// TwinCAT 3 PLC project VFDLibraryPLC
// ProgramVersion: 3.1.4023.0
// libraries:
//   Tc2_EtherCAT, * (Beckhoff Automation GmbH)
//   Tc2_Standard, * (Beckhoff Automation GmbH)
//   Tc2_System, * (Beckhoff Automation GmbH)
//   Tc2_Utilities, * (Beckhoff Automation GmbH)
//   Tc3_Module, * (Beckhoff Automation GmbH)
//   VLT_ECAT_LIB_V1_12,1.12,Danfoss Drives
// project tree:
//   DUTs/ ST_VLTParameterData.TcDUT
//   GVLs/ GVL_HMI.TcGVL
//   / PlcTask.TcTTO
//   POUs/ FB_VLTDriveControl.TcPOU, MAIN.TcPOU
// real-time tasks:
//   TASK PlcTask: cycle T#10ms, priority 20, ADS port 350
// I/O:
//   DEVICE Device 4 (EtherCAT), AmsNetId 5.24.39.150.5.1
//     Box 1 (FC-302 VLT® Automation Drive) [FC-302 VLT® Automation Drive]
// variable links:
//   (this object) <-> Device 4 (EtherCAT)/Box 1 (FC-302 VLT® Automation Drive)
//     PlcTask Inputs/MAIN.fbDriveControl.fbDriveBasic.COMM_STATUS <-> InfoData/State
//     PlcTask Inputs/MAIN.fbDriveControl.fbDriveBasic.PCDREAD.MAIN_ACTUAL_VALUE <-> Transmit PDO Parameter/1605. Main Actual Value [%]
//     PlcTask Inputs/MAIN.fbDriveControl.fbDriveBasic.PCDREAD.MOTORCURRENT <-> Transmit PDO Parameter/1614. Motor current
//     PlcTask Inputs/MAIN.fbDriveControl.fbDriveBasic.PCDREAD.STATUS_WORD <-> Transmit PDO Parameter/1603. Status Word
//     PlcTask Outputs/MAIN.fbDriveControl.fbDriveBasic.PCDWRITE.CONTROL_WORD <-> Receive PDO Parameter/1680. Fieldbus CTW 1
//     PlcTask Outputs/MAIN.fbDriveControl.fbDriveBasic.PCDWRITE.REF_VALUE <-> Receive PDO Parameter/1682. Fieldbus REF 1

CONFIGURATION VFDLibraryPLC
    RESOURCE PLC ON TwinCAT3
        TASK PlcTask(INTERVAL := T#10ms, PRIORITY := 20);
        PROGRAM MAIN WITH PlcTask : MAIN;
    END_RESOURCE
END_CONFIGURATION

// ---- DUTs/ST_VLTParameterData.TcDUT
TYPE ST_VLTParameterData :
STRUCT
	//nType		: UINT; //1 for number 2 for string.
	nRdVal		: ULINT;
	strRdVal	: STRING;
	nWrVal		: UDINT;
	strWrVal	: STRING;
END_STRUCT
END_TYPE

// ---- GVLs/GVL_HMI.TcGVL
{attribute 'qualified_only'}
VAR_GLOBAL
	bReset		: BOOL;
	bWarning	: BOOL;
	bHandOn		: BOOL;
	bOkay		: BOOL;
	bOff		: BOOL;
	bAutoOn		: BOOL;
	bAlarm		: BOOL;
	arrParamData	: ARRAY[0..99] OF ST_VLTParameterData;
	arrParamNo		: ARRAY[0..99] OF UINT;
	nParamCount	:	INT;
	bRdParams	: BOOL;
	bRdDone		: BOOL;
	bWrParams	: BOOL;
	bWrDone		: BOOL;
END_VAR

// ---- POUs/MAIN.TcPOU
PROGRAM MAIN
VAR
	fbDriveControl	: FB_VLTDriveControl;
	bEnable		: BOOL;
	bRun		: BOOL;
	nSpeed		: INT;
	bReverse	: BOOL;
	nState		: INT;
	bResetDrive	: BOOL;
	sDriveAmsNetId	: STRING := '5.24.39.150.5.1';
	nDriveAddr	: UINT := 1001;
	nAlarms		: ULINT;
	nWarnings	: ULINT;
	bRdParam	: BOOL;
	bWrParam	: BOOL;
	nParamNo	: UINT;
	nCounter	: INT;
	cbAmntRd	: UDINT;
	nParResult	: ULINT;
	fbCoERead	: FB_EcCoESdoRead;
	fbCoEWrite	: FB_EcCoESdoWrite;
	EL7411	AT %I* : UDINT;
	nCheck	: INT := 0;
END_VAR

CASE nState OF
0:
	IF(fbDriveControl.Initialize(sDriveAmsNetId,nDriveAddr)) THEN
		nState :=1;
	END_IF
1:
bEnable :=TRUE;
	IF fbDriveControl.bDriveReady AND NOT fbDriveControl.bDriveFault THEN
		nState := 2;
	END_IF
2:
	bRun	:= FALSE;
	nSpeed := 5000;
	bReverse := FALSE;
	nState := 3;
	fbCoERead(
	sNetId:= sDriveAmsNetId, 
	nSlaveAddr:= nDriveAddr, 
	tTimeout:= T#5S,
	bExecute := FALSE 
	);
	fbCoEWrite(
	sNetId:= sDriveAmsNetId, 
	nSlaveAddr:= nDriveAddr, 
	tTimeout := T#5S,
	bExecute := FALSE
	);
3: 
	
	IF GVL_HMI.bRdParams OR GVL_HMI.bWrDone THEN		
		nState := 4;
	ELSE 
		bRdParam := FALSE;
	END_IF
	
	IF GVL_HMI.bWrParams AND NOT fbDriveControl.bParBusy THEN
		nState := 6;
	ELSE
		bWrParam := FALSE;		
	END_IF
4:
	bRdParam := TRUE;
	fbCoERead.nIndex := UINT_TO_WORD(GVL_HMI.arrParamNo[nCounter]+ 16#2000);
	fbCoERead.nSubIndex := 0;
	GVL_HMI.arrParamData[nCounter].nRdVal := 0;
	fbCoERead.pDstBuf := ADR(GVL_HMI.arrParamData[nCounter].nRdVal);
	fbCoeRead.cbBufLen := SIZEOF(GVL_HMI.arrParamData[nCounter].nRdVal);

		
	nState := 5;

5:
			
		
		IF NOT fbCoERead.bBusy AND NOT fbCoERead.bError THEN
			bRdParam := FALSE;
			
			nParResult := 0;		
			IF nCounter < GVL_HMI.nParamCount - 1THEN		
				nCounter := nCounter +1;
				nState :=	4;	
			ELSE
				nCounter := 0;
				nState := 3;
				GVL_HMI.bRdParams := FALSE;
				GVL_HMI.bRdDone	:= TRUE;
				GVL_HMI.bWrDone := FALSE;
			END_IF
		END_IF
		
	IF fbCoERead.bError THEN
		IF fbCoERead.nErrId = 1795 OR fbCoERead.nErrId =1797 THEN
			GVL_HMI.arrParamData[nCounter].nRdVal := fbCoERead.nErrId;
			nCounter := nCounter +1;
		END_IF
		bRdParam:= FALSE;
		nState := 3;	
	END_IF
6:
	bWrParam := TRUE;
	fbCoEWrite.nSubIndex:= 0; 
	IF GVL_HMI.arrParamData[nCounter].nWrVal <> GVL_HMI.arrParamData[nCounter].nRdVal THEN
	fbCoEWrite.nIndex:= GVL_HMI.arrParamNo[nCounter] + 16#2000; 
	fbCoEWrite.pSrcBuf:= ADR(GVL_HMI.arrParamData[nCounter].nWrVal); 
	fbCoEWrite.cbBufLen:= SIZEOF(GVL_HMI.arrParamData[nCounter].nWrVal);	
	nState := 7;
	ELSE
		IF nCounter < GVL_HMI.nParamCount-1 THEN
			nCounter := nCounter+1;	
		ELSE
			nCounter := 0;
			nState := 3;
			GVL_HMI.bWRParams := FALSE;
			GVL_HMI.bWrDone	:= TRUE;
		END_IF
	END_IF
7:
	IF NOT fbCoEWrite.bBusy AND NOT fbCoEWrite.bError THEN
			bWrParam := FALSE;
			
			IF nCounter < GVL_HMI.nParamCount - 1THEN		
				nCounter := nCounter +1;
				nState :=	6;	
			ELSE
				nCounter := 0;
				nState := 3;
				GVL_HMI.bWRParams := FALSE;
				GVL_HMI.bWrDone	:= TRUE;
			END_IF
				
				
		END_IF
		
	IF fbCoEWrite.bError THEN
		IF fbCoEWrite.nErrId = 1795 OR fbCoEWrite.nErrId =1797 THEN
			nCounter := nCounter +1;
		END_IF
		bWrParam:= FALSE;
		nState := 3;	
	END_IF
END_CASE

fbDriveControl.DriveRun(bEnable,bRun,bReverse,nSpeed,bResetDrive);


IF NOT fbDriveControl.bDriveFault THEN
		//fbDriveControl.GetDriveDiag(nDriveAlarms =>nAlarms,nDriveWarningS => nWarnings,bAlarm =>GVL_HMI.bAlarm, bWarning => GVL_HMI.bWarning);
		IF GVL_HMI.bAlarm OR GVL_HMI.bWarning OR GVL_HMI.bReset THEN
			bResetDrive := TRUE;
		END_IF
END_IF
fbCoERead(bExecute := bRdParam,cbRead =>cbAmntRd);
fbCoEWrite(bExecute := bWrParam);
GVL_HMI.bOkay := fbDriveControl.bDriveReady;

END_PROGRAM

// ---- POUs/FB_VLTDriveControl.TcPOU
FUNCTION_BLOCK FB_VLTDriveControl
VAR_INPUT
END_VAR
VAR_OUTPUT
	bDriveReady			: BOOL;
	bDriveFault			: BOOL;
	bDriveWarning		: BOOL;
	bDriveRunning		: BOOL;
	bDriveRunOnRef		: BOOL;
	bDriveComOk			: BOOL;
	nDriveMAV			: INT;
	fDriveMtrCurrent	: REAL;
	bParBusy			: BOOL;
	bRdDone				: BOOL;
	bRdFault			: BOOL;
	nRdFaultCode		: UDINT;
	bWrDone				: BOOL;
	bWrFault			: BOOL;
	bWrFaultCode		: BOOL;
END_VAR
VAR
	fbDriveBasic		: VLT_ECAT_FC_BASIC;
	fbDriveDiag			: VLT_ECAT_FC_DIAGNOSTICS;
	fbDriveParams		: VLT_ECAT_FC_PARAM_ACCESS;
	fbEcRead			: FB_EcCoESdoRead;
	fbEcWrite			: FB_EcCoESdoWrite;
	nECode				: ULINT;
	
	nSubIndex			: BYTE;
	nRdResult			: ULINT;

	
END_VAR

METHOD DriveRun : BOOL
VAR_INPUT
	bEnable	: BOOL;
	bRun	: BOOL;
	bReverse	: BOOL;
	nSpeed	: INT;
	bReset	: BOOL;
END_VAR
fbDriveBasic(
	DRV_EN:= bEnable, 
	RUN:= bRun, 
	REVERSE:= bReverse, 
	REF_VALUE:= nSpeed, 
	RESET:= GVL_HMI.bReset, 
	READY=> bDriveReady, 
	FAULT=> bDriveFault, 
	WARNING=> bDriveWarning, 
	RUNNING=> bDriveRunning, 
	RUN_ON_REF=> bDriveRunOnRef, 
	COMM_OK=> bDriveComOk, 
	MAV=> nDriveMAV, 
	MOTORCURRENT=> fDriveMtrCurrent);
END_METHOD

METHOD GetDriveDiag : BOOL
VAR_INPUT
END_VAR
VAR_OUTPUT
	bAlarm			: BOOL;
	nDriveAlarms	: ULINT;
	bWarning		: BOOL;
	nDriveWarningS	: ULINT;
END_VAR
fbDriveDiag( 
	ALARM_1=> nDriveAlarms, 
	WARNING_1=> nDriveWarnings, 
	EMCY_CODE=> nECODE);
	
IF ndriveAlarms >0 THEN
	bAlarm := TRUE;
ELSE
	bAlarm := FALSE;
END_IF

IF nDriveWarnings >0 THEN
	bWarning	:=TRUE;
ELSE
	bWarning := FALSE;
END_IF
END_METHOD

METHOD Initialize : BOOL
VAR_INPUT
	sDriveNetID	: STRING;
	nDriveAddr	: UINT;
END_VAR
fbDriveDiag.AMS_NET_ID:= sDriveNetID;
fbDriveDiag.SLAVE_ADDR:= nDriveAddr; 
fbDriveDiag.TIMEOUT:=T#5S; 
	
fbEcRead.sNETID:= sDriveNetID; 
fbEcRead.nSlaveAddr:= nDriveAddr; 
fbEcRead.tTIMEOUT:= T#5S; 
Initialize := TRUE;
END_METHOD

{attribute 'Invoke_RPC_ENABLE' := '1'}
METHOD RdDriveParams : BOOL
VAR_INPUT
	bRdParams		: BOOL;
	nParameterNo	: UINT;
	bIsString		: BOOL;
END_VAR
VAR_OUTPUT
	nRESULT : ULINT;
	StrRESULT	: STRING;
	cbRd	: UDINT;
END_VAR

(*fbDriveParams(
	EXECUTE:= bRdParams, 
	RD_WR:= FALSE, 
	IS_STR:= bIsString, 
	PAR_NO:= nParameterNo,
	SUBINDEX := 0, 
	RD_VALUE=> nRESULT,
	STR_RD_VALUE => strRESULT,
	BUSY=> bParBusy, 
	DONE=> bRdDone, 
	FAULT=> bRdFault,
	FAULT_CODE=>nRdFaultCode);
	*)
fbEcRead(
	nSubIndex:= 0, 
	nIndex:= UINT_TO_WORD(nParameterNo + 16#2000), 
	pDstBuf:= ADR(nRdRESULT), 
	cbBufLen:= SIZEOF(nRdRESULT), 
	bExecute:= bRdParams,  
	bBusy=> bParBusy, 
	bError=> bRdFault, 
	nErrId=> nRdFaultCode, 
	cbRead=> cbRd
);
IF nRdResult >0 THEN
	nRESULT := nRdResult;
	nRdResult := 0;
END_IF
END_METHOD

METHOD WrDriveParams : BOOL
VAR_INPUT
	bWrParams		: BOOL;
	nParameterNo	: UINT;
	bIsString		: BOOL;
	
END_VAR
VAR_INST
	nWrIndex	: INT;
END_VAR
fbDriveParams(
	EXECUTE:= bWrParams, 
	RD_WR:= TRUE, 
	IS_STR:= bIsString, 
	PAR_NO:= nParameterNo,
	WR_VALUE:= GVL_HMI.arrParamData[nWrIndex].nWrVal, 
	STR_WR_VALUE:= GVL_HMI.arrParamData[nWrIndex].strWrVal, 
	BUSY=> bParBusy, 
	DONE=> bWrDone, 
	FAULT=> bWrFault);
	
IF bWrDone THEN
	nWrIndex := nWrIndex + 1;
END_IF
END_METHOD

END_FUNCTION_BLOCK
